// TIA Portal V19 export
VAR_GLOBAL   // PLC tag table "Tag table from XML_1"
   "Start Button 0" AT %I0.0 : Bool;
   "Stop Button 0" AT %I0.1 : Bool;
   "Belt Conveyor (4m) 0" AT %Q0.0 : Bool;
END_VAR
